KUKA KRL program: p01pick1.src, p01pick1.dat

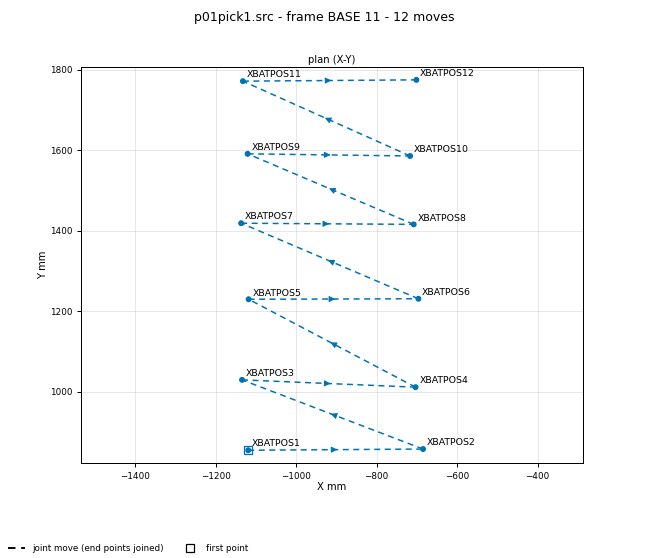
[picture p0: tool path of p01pick1.src in frame BASE 11, 12 of 13 moves have a stored position in this frame; points joined in program order, loops and branches not executed]
--- p01pick1.src ---
&ACCESS RVO1
&REL 85
&COMMENT Pick Part
&PARAM EDITMASK = *
&PARAM TEMPLATE = C:\KRC\Roboter\Template\vorgabe
&PARAM DISKPATH = KRC:\R1\Program\Sub Programs
DEF P01pick1( )
;FOLD INI
  ;FOLD BASISTECH INI
BACKJUMP=FALSE
CARTJUMP=FALSE
    GLOBAL INTERRUPT DECL 3 WHEN $STOPMESS==TRUE DO IR_STOPM ( )
    INTERRUPT ON 3
    BAS (#INITMOV,0 )
  ;ENDFOLD (BASISTECH INI)
;ENDFOLD (INI)
;================================================
; MODEL    : XXXX
; IE GROUP : XX
; STATION  : XXX
; ROBOT    : RX
; FUNCTION : pick Part in StXX
;================================================

;wait point

ACT_OV=$OV_PRO
;FOLD PTP P01waitdrop Vel=100 % PDAT1 Tool[5] Base[0];%{PE}%R 8.3.48,%MKUKATPBASIS,%CMOVE,%VPTP,%P 1:PTP, 2:P01waitdrop, 3:, 5:100, 7:PDAT1
$BWDSTART=FALSE
PDAT_ACT=PPDAT1
FDAT_ACT=FP01waitdrop
BAS(#PTP_PARAMS,100)
PTP XP01waitdrop
;ENDFOLD


WAIT FOR ($IN[54]==TRUE) OR ($IN[1]==TRUE)

IF $in[54]==TRUE THEN
   bombero ( )               ; PICK In Station XX
   ENDIF
;IF FALSE THEN
;FOLD TYPE INFO

IF (I_TYPE_INFO<100)THEN
POSBAT=I_TYPE_INFO
PISO=0
ENDIF
IF (I_TYPE_INFO>100) AND (I_TYPE_INFO<200)THEN
POSBAT=I_TYPE_INFO-100
PISO=1
ENDIF
IF (I_TYPE_INFO>200) AND (I_TYPE_INFO<300)THEN
POSBAT=I_TYPE_INFO-200
PISO=2
ENDIF

;Guarda dato para Tciclo
ALT_TC=PISO

O_TYPE_REQ=FALSE

;ENDFOLD

;Para timer durante area req
$TIMER_STOP[7]=TRUE

;Wait For Area / Goto Safety / Return To Home
;FOLD Fordtech.Area_Req Area Request: 1, Safety Position: 0, Return To Home: 0;%{PE}%MKUKATPUSER

Area_Req (1,0,0)
IF I_RETHP AND (0 <> 0) AND ($IN_HOME == TRUE) THEN
  GOTO PEXIT
ENDIF

;ENDFOLD

;ENDIF
;cils_init()

;Arranca timer despues de area req
$TIMER_STOP[7]=FALSE


;FOLD ALTUA BASE
level1=PISO
BASE_DATA[11]=BASE_DATA[13]
BASE_DATA[11].Z=BASE_DATA[11].Z+(ALTURA1*LEVEL1)

;ENDFOLD

;Guarda pos bateria para Tciclo
POS_BAT_TC=POSBAT

SWITCH POSBAT ;posicion bateria

CASE 1

;POS FOTO BATERIA 1
;FOLD PTP BATPOS1 Vel=100 % M Tool[5]:Gripper_empty Base[11];%{PE}%R 8.3.48,%MKUKATPBASIS,%CMOVE,%VPTP,%P 1:PTP, 2:BATPOS1, 3:, 5:100, 7:M
$BWDSTART=FALSE
PDAT_ACT=PM
FDAT_ACT=FBATPOS1
BAS(#PTP_PARAMS,100)
PTP XBATPOS1
;ENDFOLD
WAIT SEC 0.3

CASE 2

;POS FOTO BATERIA 2
;FOLD PTP BATPOS2 Vel=100 % M Tool[5]:Gripper_empty Base[11];%{PE}%R 8.3.48,%MKUKATPBASIS,%CMOVE,%VPTP,%P 1:PTP, 2:BATPOS2, 3:, 5:100, 7:M
$BWDSTART=FALSE
PDAT_ACT=PM
FDAT_ACT=FBATPOS2
BAS(#PTP_PARAMS,100)
PTP XBATPOS2
;ENDFOLD
WAIT SEC 0.3

CASE 3

;POS FOTO BATERIA 3
;FOLD PTP BATPOS3 Vel=100 % M Tool[5]:Gripper_empty Base[11];%{PE}%R 8.3.48,%MKUKATPBASIS,%CMOVE,%VPTP,%P 1:PTP, 2:BATPOS3, 3:, 5:100, 7:M
$BWDSTART=FALSE
PDAT_ACT=PM
FDAT_ACT=FBATPOS3
BAS(#PTP_PARAMS,100)
PTP XBATPOS3
;ENDFOLD
WAIT SEC 0.3

CASE 4

;POS FOTO BATERIA 4
;FOLD PTP BATPOS4 Vel=100 % M Tool[5]:Gripper_empty Base[11];%{PE}%R 8.3.48,%MKUKATPBASIS,%CMOVE,%VPTP,%P 1:PTP, 2:BATPOS4, 3:, 5:100, 7:M
$BWDSTART=FALSE
PDAT_ACT=PM
FDAT_ACT=FBATPOS4
BAS(#PTP_PARAMS,100)
PTP XBATPOS4
;ENDFOLD
WAIT SEC 0.3

CASE 5

;POS FOTO BATERIA 5
;FOLD PTP BATPOS5 Vel=100 % M Tool[5]:Gripper_empty Base[11];%{PE}%R 8.3.48,%MKUKATPBASIS,%CMOVE,%VPTP,%P 1:PTP, 2:BATPOS5, 3:, 5:100, 7:M
$BWDSTART=FALSE
PDAT_ACT=PM
FDAT_ACT=FBATPOS5
BAS(#PTP_PARAMS,100)
PTP XBATPOS5
;ENDFOLD
WAIT SEC 0.3

CASE 6

;POS FOTO BATERIA 6
;FOLD PTP BATPOS6 Vel=100 % M Tool[5]:Gripper_empty Base[11];%{PE}%R 8.3.48,%MKUKATPBASIS,%CMOVE,%VPTP,%P 1:PTP, 2:BATPOS6, 3:, 5:100, 7:M
$BWDSTART=FALSE
PDAT_ACT=PM
FDAT_ACT=FBATPOS6
BAS(#PTP_PARAMS,100)
PTP XBATPOS6
;ENDFOLD
WAIT SEC 0.3

CASE 7

;POS FOTO BATERIA 7
;FOLD PTP BATPOS7 Vel=100 % M Tool[5]:Gripper_empty Base[11];%{PE}%R 8.3.48,%MKUKATPBASIS,%CMOVE,%VPTP,%P 1:PTP, 2:BATPOS7, 3:, 5:100, 7:M
$BWDSTART=FALSE
PDAT_ACT=PM
FDAT_ACT=FBATPOS7
BAS(#PTP_PARAMS,100)
PTP XBATPOS7
;ENDFOLD
WAIT SEC 0.3

CASE 8

;POS FOTO BATERIA 8
;FOLD PTP BATPOS8 Vel=100 % M Tool[5]:Gripper_empty Base[11];%{PE}%R 8.3.48,%MKUKATPBASIS,%CMOVE,%VPTP,%P 1:PTP, 2:BATPOS8, 3:, 5:100, 7:M
$BWDSTART=FALSE
PDAT_ACT=PM
FDAT_ACT=FBATPOS8
BAS(#PTP_PARAMS,100)
PTP XBATPOS8
;ENDFOLD
WAIT SEC 0.3

CASE 9

;POS FOTO BATERIA 9
;FOLD PTP BATPOS9 Vel=100 % M Tool[5]:Gripper_empty Base[11];%{PE}%R 8.3.48,%MKUKATPBASIS,%CMOVE,%VPTP,%P 1:PTP, 2:BATPOS9, 3:, 5:100, 7:M
$BWDSTART=FALSE
PDAT_ACT=PM
FDAT_ACT=FBATPOS9
BAS(#PTP_PARAMS,100)
PTP XBATPOS9
;ENDFOLD
WAIT SEC 0.3

CASE 10

;POS FOTO BATERIA 10
;FOLD PTP BATPOS10 Vel=100 % M Tool[5]:Gripper_empty Base[11];%{PE}%R 8.3.48,%MKUKATPBASIS,%CMOVE,%VPTP,%P 1:PTP, 2:BATPOS10, 3:, 5:100, 7:M
$BWDSTART=FALSE
PDAT_ACT=PM
FDAT_ACT=FBATPOS10
BAS(#PTP_PARAMS,100)
PTP XBATPOS10
;ENDFOLD
WAIT SEC 0.3

CASE 11

;POS FOTO BATERIA 11
;FOLD PTP BATPOS11 Vel=100 % M Tool[5]:Gripper_empty Base[11];%{PE}%R 8.3.48,%MKUKATPBASIS,%CMOVE,%VPTP,%P 1:PTP, 2:BATPOS11, 3:, 5:100, 7:M
$BWDSTART=FALSE
PDAT_ACT=PM
FDAT_ACT=FBATPOS11
BAS(#PTP_PARAMS,100)
PTP XBATPOS11
;ENDFOLD
WAIT SEC 0.3
;ACT_OV=$OV_PRO
;$OV_PRO=10
CASE 12

;POS FOTO BATERIA 12
;FOLD PTP BATPOS12 Vel=100 % M Tool[5]:Gripper_empty Base[11];%{PE}%R 8.3.48,%MKUKATPBASIS,%CMOVE,%VPTP,%P 1:PTP, 2:BATPOS12, 3:, 5:100, 7:M
$BWDSTART=FALSE
PDAT_ACT=PM
FDAT_ACT=FBATPOS12
BAS(#PTP_PARAMS,100)
PTP XBATPOS12
;ENDFOLD
WAIT SEC 0.3
;ACT_OV=$OV_PRO
;$OV_PRO=10
CASE 13

;CARTON
P01pick1_2corr()
P01drop2()

CARTJUMP=TRUE
GOTO PEXIT

DEFAULT
;ESTO NO DEBERIA HABER OCURRIDO, KEEP CALM
WAIT FOR FALSE

ENDSWITCH

$ACT_BASE=0
$ACT_TOOL=0

panpick()

$OV_PRO=ACT_OV
;fold provisional para pruebas
M_TYPE_INFO=M_TYPE_INFO+1
;endfold



;Release Area 1

;FOLD SYN OUT 17 'Area Release 1' State=TRUE at START Delay=0 ms;%{PE}%R 8.3.48,%MKUKATPBASIS,%COUT,%VSYNOUT,%P 2:17, 3:Area Release 1, 5:TRUE, 7:0, 9:0, 12:0
TRIGGER WHEN DISTANCE=0 DELAY=0 DO $OUT[17]=TRUE
;ENDFOLD
;Jump Adress
PEXIT:

;Guarda TC por cada array cogido y carton para rack1
;FOLD Guarda_TC
;ALT_TC es 1, 2, o 3
;POS_BAT_TC va de 1 a 12 y 13 para carton
$TIMER_STOP[7]=TRUE
IF POS_BAT_TC < 13 THEN
   INDICE_PICK=POS_BAT_TC+(12*ALT_TC)
   TC_PICK_RACK1[INDICE_PICK]=$TIMER[7]
ENDIF

IF (POS_BAT_TC==13) THEN
   IF (ALT_TC==2) THEN
      TC_CARTON[1]=$TIMER[7]
   ENDIF
   IF (ALT_TC==1) THEN
      TC_CARTON[2]=$TIMER[7]
   ENDIF
ENDIF

;ENDFOLD

END

--- p01pick1.dat ---
&ACCESS RVO1
&REL 85
&COMMENT Pick Part
&PARAM EDITMASK = *
&PARAM TEMPLATE = C:\KRC\Roboter\Template\vorgabe
&PARAM DISKPATH = KRC:\R1\Program\Sub Programs
DEFDAT  p01pick1

EXT  BAS (BAS_COMMAND  :IN,REAL  :IN )
DECL INT SUCCESS
;******************************
;*     E6POS Declarations     *
;******************************

DECL E6POS XP01WAITREQ2={X 2157.35596,Y -301.755188,Z 2852.14893,A -15.8183,B 72.8074417,C -9.82211304,S 2,T 34,E1 0.0,E2 0.0,E3 0.0,E4 0.0,E5 0.0,E6 0.0}
DECL E6POS XP10={X 2411.43896,Y 1748.73096,Z -1095.62903,A -177.692307,B -16.9195194,C 42.7874298,S 2,T 34,E1 0.0,E2 0.0,E3 0.0,E4 0.0,E5 0.0,E6 0.0}
DECL E6POS XP20={X 1670.59900,Y -157.831207,Z 2354.64209,A -15.8183,B 72.8074417,C -9.82211304,S 2,T 34,E1 0.0,E2 0.0,E3 0.0,E4 0.0,E5 0.0,E6 0.0}
DECL E6POS XP30={X 1670.59900,Y -157.831207,Z 2354.64209,A -15.8183,B 72.8074417,C -9.82211304,S 2,T 34,E1 0.0,E2 0.0,E3 0.0,E4 0.0,E5 0.0,E6 0.0}
DECL E6POS XDROP_POS={X 1670.59900,Y -157.831207,Z 2354.64209,A -15.8183,B 72.8074417,C -9.82211304,S 2,T 34,E1 0.0,E2 0.0,E3 0.0,E4 0.0,E5 0.0,E6 0.0}
DECL E6POS XP40={X 2411.43896,Y 1748.73096,Z -1095.62903,A -177.692307,B -16.9195194,C 42.7874298,S 2,T 34,E1 0.0,E2 0.0,E3 0.0,E4 0.0,E5 0.0,E6 0.0}
DECL E6POS XP50={X 2411.43896,Y 1748.73096,Z -1095.62903,A -177.692307,B -16.9195194,C 42.7874298,S 2,T 34,E1 0.0,E2 0.0,E3 0.0,E4 0.0,E5 0.0,E6 0.0}
DECL E6POS XP01WAITREL2={X 2411.43896,Y 1748.73096,Z -1095.62903,A -177.692307,B -16.9195194,C 42.7874298,S 2,T 34,E1 0.0,E2 0.0,E3 0.0,E4 0.0,E5 0.0,E6 0.0}

;******************************
;*     FDAT Declarations      *
;******************************

DECL FDAT FP01WAITREQ2={TOOL_NO 12,BASE_NO 0,IPO_FRAME #BASE}
DECL FDAT FP10={TOOL_NO 12,BASE_NO 0,IPO_FRAME #TCP}
DECL FDAT FP20={TOOL_NO 12,BASE_NO 0,IPO_FRAME #TCP}
DECL FDAT FP30={TOOL_NO 12,BASE_NO 0,IPO_FRAME #TCP}
DECL FDAT FDROP_POS={TOOL_NO 12,BASE_NO 0,IPO_FRAME #TCP}
DECL FDAT FP40={TOOL_NO 12,BASE_NO 0,IPO_FRAME #TCP}
DECL FDAT FP50={TOOL_NO 12,BASE_NO 0,IPO_FRAME #TCP}
DECL FDAT FP01WAITREL2={TOOL_NO 12,BASE_NO 0,IPO_FRAME #TCP}

;******************************
;*  PDAT & LDAT Declarations  *
;******************************

DECL PDAT PH={VEL 100.000,ACC 100.000,APO_DIST 100.000,APO_MODE #CDIS,GEAR_JERK 100.000,EXAX_IGN 0}

DECL MODULEPARAM_T LAST_TP_PARAMS={PARAMS[] "FORDTECH.P_AREA_REQ=2; FORDTECH.P_SAFETY_POS=0; FORDTECH.P_RET=0; Kuka.VelocityFieldEnabled=True; Kuka.ColDetectFieldEnabled=True; Kuka.MovementParameterFieldEnabled=True; Kuka.IsAngleEnabled=False; Kuka.PointName=P01Waitdrop; Kuka.FrameData.base_no=0; Kuka.FrameData.tool_no=5; Kuka.FrameData.ipo_frame=#BASE; Kuka.isglobalpoint=False; Kuka.MoveDataPtpName=H; Kuka.MovementDataPdat.apo_mode=#CDIS; Kuka.MovementDataPdat.apo_dist=100; Kuka.MovementData.vel=100; Kuka.MovementData.acc=100; Kuka.MovementData.exax_ign=0; Kuka.VelocityPtp=100; Kuka.BlendingEnabled=False; Kuka.APXEnabled=False; Kuka.CurrentCDSetIndex=0; Kuka.FrameData.point2=                         "}
DECL E6POS XP01Waitdrop={X 290.951233,Y 816.177124,Z 1275.55042,A -86.9976196,B 22.0779018,C -179.006119,S 6,T 27,E1 0.0,E2 0.0,E3 0.0,E4 0.0,E5 0.0,E6 0.0}
DECL FDAT FP01Waitdrop={TOOL_NO 5,BASE_NO 0,IPO_FRAME #BASE,POINT2[] " ",TQ_STATE FALSE}
DECL E6POS XBATPOS1={X -1118.94214,Y 855.193665,Z 1101.31165,A -87.0149307,B 22.0764637,C -179.006195,S 6,T 27,E1 0.0,E2 0.0,E3 0.0,E4 0.0,E5 0.0,E6 0.0}
DECL FDAT FBATPOS1={TOOL_NO 5,BASE_NO 11,IPO_FRAME #BASE,POINT2[] " ",TQ_STATE FALSE}
DECL E6POS XBATPOS2={X -684.757935,Y 858.192078,Z 1101.07874,A -87.0149612,B 22.0764923,C -179.006210,S 6,T 27,E1 0.0,E2 0.0,E3 0.0,E4 0.0,E5 0.0,E6 0.0}
DECL FDAT FBATPOS2={TOOL_NO 5,BASE_NO 11,IPO_FRAME #BASE,POINT2[] " "}
DECL E6POS XBATPOS3={X -1134.34216,Y 1030.01428,Z 1104.29102,A -87.0149307,B 22.0764618,C -179.006195,S 6,T 27,E1 0.0,E2 0.0,E3 0.0,E4 0.0,E5 0.0,E6 0.0}
DECL FDAT FBATPOS3={TOOL_NO 5,BASE_NO 11,IPO_FRAME #BASE,POINT2[] " "}
DECL E6POS XBATPOS4={X -703.399292,Y 1011.80255,Z 1100.54785,A -87.0149307,B 22.0764656,C -179.006195,S 6,T 27,E1 0.0,E2 0.0,E3 0.0,E4 0.0,E5 0.0,E6 0.0}
DECL FDAT FBATPOS4={TOOL_NO 5,BASE_NO 11,IPO_FRAME #BASE,POINT2[] " "}
DECL E6POS XBATPOS5={X -1117.99915,Y 1230.22937,Z 1089.50244,A -87.0149307,B 22.0764637,C -179.006195,S 6,T 27,E1 0.0,E2 0.0,E3 0.0,E4 0.0,E5 0.0,E6 0.0}
DECL FDAT FBATPOS5={TOOL_NO 5,BASE_NO 11,IPO_FRAME #BASE,POINT2[] " "}
DECL E6POS XBATPOS6={X -696.272949,Y 1231.45142,Z 1087.81201,A -86.9321365,B 22.0656681,C -178.785858,S 6,T 27,E1 0.0,E2 0.0,E3 0.0,E4 0.0,E5 0.0,E6 0.0}
DECL FDAT FBATPOS6={TOOL_NO 5,BASE_NO 11,IPO_FRAME #BASE,POINT2[] " "}
DECL E6POS XBATPOS7={X -1136.56091,Y 1419.10437,Z 1097.47314,A -87.0149307,B 22.0764637,C -179.006195,S 6,T 27,E1 0.0,E2 0.0,E3 0.0,E4 0.0,E5 0.0,E6 0.0}
DECL FDAT FBATPOS7={TOOL_NO 5,BASE_NO 11,IPO_FRAME #BASE,POINT2[] " "}
DECL E6POS XBATPOS8={X -707.989807,Y 1416.22681,Z 1102.96265,A -87.0148773,B 22.0764618,C -179.006042,S 6,T 27,E1 0.0,E2 0.0,E3 0.0,E4 0.0,E5 0.0,E6 0.0}
DECL FDAT FBATPOS8={TOOL_NO 5,BASE_NO 11,IPO_FRAME #BASE,POINT2[] " "}
DECL E6POS XBATPOS9={X -1120.45471,Y 1591.43530,Z 1098.53064,A -87.0149307,B 22.0764637,C -179.006195,S 6,T 27,E1 0.0,E2 0.0,E3 0.0,E4 0.0,E5 0.0,E6 0.0}
DECL FDAT FBATPOS9={TOOL_NO 5,BASE_NO 11,IPO_FRAME #BASE,POINT2[] " "}
DECL E6POS XBATPOS10={X -716.971619,Y 1586.09741,Z 1104.78284,A -87.0149307,B 22.0764637,C -179.006195,S 6,T 27,E1 0.0,E2 0.0,E3 0.0,E4 0.0,E5 0.0,E6 0.0}
DECL FDAT FBATPOS10={TOOL_NO 5,BASE_NO 11,IPO_FRAME #BASE,POINT2[] " "}
DECL E6POS XBATPOS11={X -1132.20166,Y 1771.93982,Z 1091.64111,A -87.0149307,B 22.0764694,C -179.006195,S 6,T 27,E1 0.0,E2 0.0,E3 0.0,E4 0.0,E5 0.0,E6 0.0}
DECL FDAT FBATPOS11={TOOL_NO 5,BASE_NO 11,IPO_FRAME #BASE,POINT2[] " "}
DECL E6POS XBATPOS12={X -701.332825,Y 1775.19885,Z 1100.71460,A -86.9886169,B 22.0730648,C -178.936188,S 6,T 27,E1 0.0,E2 0.0,E3 0.0,E4 0.0,E5 0.0,E6 0.0}
DECL FDAT FBATPOS12={TOOL_NO 5,BASE_NO 11,IPO_FRAME #BASE,POINT2[] " "}
DECL BASIS_SUGG_T LAST_BASIS={POINT1[] "P02Waitdrop             ",POINT2[] "P02Waitdrop             ",CP_PARAMS[] "CPDAT0                  ",PTP_PARAMS[] "PDAT15                  ",CONT[] "                        ",CP_VEL[] "2.0                     ",PTP_VEL[] "100                     ",SYNC_PARAMS[] "SYNCDAT                 ",SPL_NAME[] "S0                      ",A_PARAMS[] "ADAT0                   "}
DECL PDAT PPDAT1={VEL 100.000,ACC 100.000,APO_DIST 100.000,GEAR_JERK 50.0000,EXAX_IGN 0}
DECL PDAT PPDAT2={VEL 100.000,ACC 100.000,APO_DIST 100.000,GEAR_JERK 50.0000,EXAX_IGN 0}
DECL PDAT PPDAT3={VEL 100.000,ACC 100.000,APO_DIST 100.000,GEAR_JERK 50.0000,EXAX_IGN 0}
DECL PDAT PPDAT4={VEL 100.000,ACC 100.000,APO_DIST 100.000,GEAR_JERK 50.0000,EXAX_IGN 0}
DECL PDAT PPDAT5={VEL 100.000,ACC 100.000,APO_DIST 100.000,GEAR_JERK 50.0000,EXAX_IGN 0}
DECL PDAT PPDAT6={VEL 100.000,ACC 100.000,APO_DIST 100.000,GEAR_JERK 50.0000,EXAX_IGN 0}
DECL PDAT PPDAT7={VEL 100.000,ACC 100.000,APO_DIST 100.000,GEAR_JERK 50.0000,EXAX_IGN 0}
DECL PDAT PPDAT8={VEL 100.000,ACC 100.000,APO_DIST 100.000,GEAR_JERK 50.0000,EXAX_IGN 0}
DECL PDAT PPDAT9={VEL 100.000,ACC 100.000,APO_DIST 100.000,GEAR_JERK 50.0000,EXAX_IGN 0}
DECL PDAT PPDAT10={VEL 100.000,ACC 100.000,APO_DIST 100.000,GEAR_JERK 50.0000,EXAX_IGN 0}
DECL PDAT PPDAT11={VEL 100.000,ACC 100.000,APO_DIST 100.000,GEAR_JERK 50.0000,EXAX_IGN 0}
DECL PDAT PPDAT12={VEL 100.000,ACC 100.000,APO_DIST 100.000,GEAR_JERK 50.0000,EXAX_IGN 0}
DECL PDAT PPDAT13={VEL 100.000,ACC 100.000,APO_DIST 100.000,GEAR_JERK 50.0000,EXAX_IGN 0}
DECL PDAT PPDAT14={VEL 100.000,ACC 100.000,APO_DIST 100.000,APO_MODE #CDIS,GEAR_JERK 50.0000,EXAX_IGN 0}
DECL E6POS XP02WAITDROP={X 442.124359,Y -682.465210,Z 1416.05603,A -171.206314,B 14.8656197,C -154.747955,S 6,T 26,E1 0.0,E2 0.0,E3 0.0,E4 0.0,E5 0.0,E6 0.0}
DECL FDAT FP02Waitdrop={TOOL_NO 5,BASE_NO 0,IPO_FRAME #BASE,POINT2[] " ",TQ_STATE FALSE}
DECL PDAT PPDAT15={VEL 100.000,ACC 100.000,APO_DIST 100.000,GEAR_JERK 50.0000,EXAX_IGN 0}
DECL PDAT PM={VEL 100.000,ACC 50.0000,APO_DIST 100.000,GEAR_JERK 50.0000,EXAX_IGN 0}
ENDDAT
